FUNCTION_BLOCK FB_ProcessingState IMPLEMENTS I_State
VAR_INPUT
END_VAR
VAR_OUTPUT
END_VAR
VAR
	pfbStateMachine			:POINTER TO FB_StateMachine;
END_VAR

{warning 'Add property implementation'}
PROPERTY CurrentState : STRING
GET
CurrentState := 'Processing ...';
END_GET
END_PROPERTY

{warning 'Add method implementation '}
METHOD ErrorGone
// nothin happens
END_METHOD

{warning 'Add method implementation '}
METHOD ErrorOccured
pfbStateMachine^.SetState(pfbStateMachine^.NotReadyState);
END_METHOD

//FB_Init is always available implicitly and it is used primarily for initialization.
//The return value is not evaluated. For a specific influence, you can also declare the
//methods explicitly and provide additional code there with the standard initialization
//code. You can evaluate the return value.
METHOD FB_Init: BOOL
VAR_INPUT
    bInitRetains: BOOL; // TRUE: the retain variables are initialized (reset warm / reset cold)
    bInCopyCode: BOOL;  // TRUE: the instance will be copied to the copy code afterward (online change)   
	pfbStateMachine	:POINTER TO FB_StateMachine;
END_VAR
THIS^.pfbStateMachine := pfbStateMachine;
END_METHOD

{warning 'Add method implementation '}
METHOD StartProcess
// nothin happens
END_METHOD

{warning 'Add method implementation '}
METHOD StopProcess
pfbStateMachine^.SetState(pfbStateMachine^.ReadyState);
END_METHOD

END_FUNCTION_BLOCK

(* stored: Version 1.1.0.1
   POU FB_ProcessingState: Id {fc39f885-8644-4189-a52a-a3c8257417f7}, SpecialFunc None
   Property CurrentState: Id {5e0f5c70-ae9a-4750-ae74-73a4cfcaa811}
   Get Get: Id {9f3f9607-cd4f-48c7-9f3b-3b40cebe90e7}
   Method ErrorGone: Id {e5e31978-fb5e-49a4-a007-14bc4514c2ec}
   Method ErrorOccured: Id {cb3d3270-6be3-44bf-a8be-7e88dc56f32d}
   Method FB_Init: Id {57629abe-9bb8-4677-9680-27374c3b48d7}
   Method StartProcess: Id {9bdaad99-5ffc-4145-b813-631038332437}
   Method StopProcess: Id {0c44b252-aea8-4209-8ab3-10889726ad81} *)
